TYPE TcoCvirII_Control :
STRUCT
	{attribute addProperty Name "<#Cycle bit 1#>"}
	CycleBit1 : BOOL;
	{attribute addProperty Name "<#Cycle bit 2#>"}
	CycleBit2 : BOOL;
	{attribute addProperty Name "<#Cycle bit 4#>"}
	CycleBit4 : BOOL;
	{attribute addProperty Name "<#Spindle validation#>"}
	SpindleValidation : BOOL;
	{attribute addProperty Name "<#Error acknowledge#>"}
	ErrorAck : BOOL;
	{attribute addProperty Name "<#Start#>"}
	StartCycle : BOOL;
	{attribute addProperty Name "<#Direction#>"}
	Direction : BOOL;
	{attribute addProperty Name "<#Reset#>"}
	Reset : BOOL;
END_STRUCT
END_TYPE

(* stored: Version 1.1.0.1
   DUT TcoCvirII_Control: Id {b5806dfb-66bd-4a68-b7c7-788534c9d424} *)
